KUKA KRL program: PickEsteira.src, PickEsteira.dat

--- PickEsteira.src ---
&ACCESS RVO1
&REL 243
&PARAM DISKPATH = KRC:\R1\Program\40293_Furukawa\Pick
DEF PickEsteira ( )
   ;FOLD INI;%{PE}
      ;FOLD BASISTECH INI
         GLOBAL INTERRUPT DECL 3 WHEN $STOPMESS==TRUE DO IR_STOPM ( )
         INTERRUPT ON 3
         BAS (#INITMOV,0 )
      ;ENDFOLD (BASISTECH INI)
      ;FOLD USER INI
         ;Make your modifications here

      ;ENDFOLD (USER INI)
   ;ENDFOLD (INI)
   ConfGarra_nowait()

   ;FOLD CONFIGURACOES DE MOVIMENTO
      $VEL.CP = 2.5
      $ACC.CP = 8
      $APO.CVEL = 80
      $APO.CPTP = 80
      $APO.CDIS = 20
      ;Base e Tool
      $TOOL = TOOL_DATA[1]
      $BASE = $NULLFRAME
   ;ENDFOLD

   ;configura o mesmo X  e Y do Xpick_esteira_1
   Xpick_esteira_2.X = Xpick_esteira_1.X
   Xpick_esteira_3.X = Xpick_esteira_1.X

   Xpick_esteira_2.Z = Xpick_esteira_1.Z
   Xpick_esteira_3.Z = Xpick_esteira_1.Z

   SWITCH PickOp
      CASE 1
         XAPP1PICK = Xpick_esteira_1
         XSAIPICK  = Xpick_esteira_1
      CASE 2
         XAPP1PICK = Xpick_esteira_2
         XSAIPICK  = Xpick_esteira_3
   ENDSWITCH

   XAPP1PICK.Z = ALTURAPICK
   XSAIPICK.Z  = ALTURAPICK

   ;APROXIMA TOPO
   PTP XAPP1PICK C_DIS

   ;CONFIGURA GARRA
   AbreGarra()
   ;ConfGarra_Wait()

   ;PONTO DE PICK
   SWITCH PickOp
      CASE 1
         ;FOLD LIN pick_esteira_1 Vel=2 m/s CPDAT1 Tool[1]:GarraUniversal Base[0] ;%{PE}
            ;FOLD Parameters ;%{h}
               ;Params IlfProvider=kukaroboter.basistech.inlineforms.movement.old; Kuka.IsGlobalPoint=False; Kuka.PointName=pick_esteira_1; Kuka.BlendingEnabled=False; Kuka.MoveDataName=CPDAT1; Kuka.VelocityPath=2; Kuka.CurrentCDSetIndex=0; Kuka.MovementParameterFieldEnabled=True; IlfCommand=LIN
            ;ENDFOLD
            $BWDSTART = FALSE
            LDAT_ACT = LCPDAT1_esteira
            FDAT_ACT = Fpick_esteira_1
            BAS(#CP_PARAMS, 2.0)
            SET_CD_PARAMS (0)
            LIN Xpick_esteira_1
         ;ENDFOLD
      CASE 2
;FOLD LIN pick_esteira_2 CONT Vel=2 m/s CPDAT2 Tool[1]:GarraUniversal Base[0] ;%{PE}
;FOLD Parameters ;%{h}
;Params IlfProvider=kukaroboter.basistech.inlineforms.movement.old; Kuka.IsGlobalPoint=False; Kuka.PointName=pick_esteira_2; Kuka.BlendingEnabled=True; Kuka.MoveDataName=CPDAT2; Kuka.VelocityPath=2; Kuka.CurrentCDSetIndex=0; Kuka.MovementParameterFieldEnabled=True; IlfCommand=LIN
;ENDFOLD
$BWDSTART = FALSE
LDAT_ACT = LCPDAT2
FDAT_ACT = Fpick_esteira_2
BAS(#CP_PARAMS, 2.0)
SET_CD_PARAMS (0)
LIN Xpick_esteira_2 C_Dis C_Dis
;ENDFOLD

         ;FOLD LIN pick_esteira_3 Vel=2 m/s CPDAT2 Tool[1]:GarraUniversal Base[0] ;%{PE}
            ;FOLD Parameters ;%{h}
               ;Params IlfProvider=kukaroboter.basistech.inlineforms.movement.old; Kuka.IsGlobalPoint=False; Kuka.PointName=pick_esteira_3; Kuka.BlendingEnabled=False; Kuka.MoveDataName=CPDAT2; Kuka.VelocityPath=2; Kuka.CurrentCDSetIndex=0; Kuka.MovementParameterFieldEnabled=True; IlfCommand=LIN
            ;ENDFOLD
            $BWDSTART = FALSE
            LDAT_ACT = LCPDAT2_esteira
            FDAT_ACT = Fpick_esteira_3
            BAS(#CP_PARAMS, 2.0)
            SET_CD_PARAMS (0)
            LIN Xpick_esteira_3
         ;ENDFOLD
   ENDSWITCH

   ;Fecha Garra
   FechaGarra()

   ;LIN XSAIPICK C_DIS C_DIS

END

--- PickEsteira.dat ---
&ACCESS RVO1
&REL 243
&PARAM DISKPATH = KRC:\R1\Program\40293_Furukawa\Pick
DEFDAT  PICKESTEIRA PUBLIC
DECL E6POS XAPP1PICK={X 1810.00,Y 331.540924,Z 205.000,A -89.9933853,B -1.07773711E-14,C -180.000,S 2,T 2,E1 0.0,E2 0.0,E3 0.0,E4 0.0,E5 0.0,E6 0.0}
DECL E6POS XAPP2PICK={X 1839.57971,Y 331.540924,Z -199.292,A -89.9933853,B -1.07773711E-14,C -180.000,S 2,T 2,E1 0.0,E2 0.0,E3 0.0,E4 0.0,E5 0.0,E6 0.0}
DECL E6POS XPICK={X 1839.57971,Y -502.858154,Z -210.581238,A -89.9924088,B -1.01663605E-13,C -180.000,S 2,T 2,E1 0.0,E2 0.0,E3 0.0,E4 0.0,E5 0.0,E6 0.0}
DECL E6POS XSAIPICK={X 1810.00,Y 331.540924,Z 205.000,A -89.9933853,B -1.07773711E-14,C -180.000,S 2,T 2,E1 0.0,E2 0.0,E3 0.0,E4 0.0,E5 0.0,E6 0.0}
;pontos exportados de FURUKAWA
DECL LDAT LCPDAT1_esteira={VEL 2.00000,ACC 100.000,APO_DIST 500.000,APO_FAC 50.0000,AXIS_VEL 100.000,AXIS_ACC 100.000,ORI_TYP #VAR,CIRC_TYP #BASE,JERK_FAC 50.0000,GEAR_JERK 100.000,EXAX_IGN 0}
DECL LDAT LCPDAT2_esteira={VEL 2.00000,ACC 100.000,APO_DIST 500.000,APO_FAC 50.0000,AXIS_VEL 100.000,AXIS_ACC 100.000,ORI_TYP #VAR,CIRC_TYP #BASE,JERK_FAC 50.0000,GEAR_JERK 100.000,EXAX_IGN 0}
DECL GLOBAL E6POS Xpick_esteira_1={X 1810.00,Y 331.540924,Z -199.292,A -89.9933853,B -1.07773711E-14,C -180.000,S 2,T 2,E1 0.0,E2 0.0,E3 0.0,E4 0.0,E5 0.0,E6 0.0}
DECL FDAT Fpick_esteira_1={TOOL_NO 1,BASE_NO 0,IPO_FRAME #BASE,POINT2[] " "}
DECL E6POS Xpick_esteira_2={X 1810.00,Y -502.858154,Z -199.292,A -89.9924088,B -1.01663605E-13,C -180.000,S 2,T 2,E1 0.0,E2 0.0,E3 0.0,E4 0.0,E5 0.0,E6 0.0}
DECL FDAT Fpick_esteira_2={TOOL_NO 1,BASE_NO 0,IPO_FRAME #BASE,POINT2[] " "}
DECL E6POS Xpick_esteira_3={X 1810.00,Y -615.344604,Z -199.292,A -89.9924088,B 1.60590833E-13,C 180.000,S 2,T 2,E1 0.0,E2 0.0,E3 0.0,E4 0.0,E5 0.0,E6 0.0}
DECL FDAT Fpick_esteira_3={TOOL_NO 1,BASE_NO 0,IPO_FRAME #BASE,POINT2[] " "}
DECL LDAT LCPDAT2={VEL 2.00000,ACC 100.000,APO_DIST 500.000,APO_FAC 50.0000,AXIS_VEL 100.000,AXIS_ACC 100.000,ORI_TYP #VAR,CIRC_TYP #BASE,JERK_FAC 50.0000,GEAR_JERK 100.000,EXAX_IGN 0}
DECL MODULEPARAM_T LAST_TP_PARAMS={PARAMS[] "Kuka.PointName=pick_esteira_2; Kuka.FrameData.base_no=0; Kuka.FrameData.tool_no=1; Kuka.FrameData.ipo_frame=#BASE; Kuka.FrameData.point2=; Kuka.isglobalpoint=False; Kuka.MoveDataName=CPDAT2; Kuka.MovementData.apo_fac=50; Kuka.MovementData.apo_dist=500; Kuka.MovementData.axis_acc=100; Kuka.MovementData.axis_vel=100; Kuka.MovementData.circ_typ=#BASE; Kuka.MovementData.jerk_fac=50; Kuka.MovementData.ori_typ=#VAR; Kuka.MovementData.vel=2; Kuka.MovementData.acc=100; Kuka.MovementData.exax_ign=0; Kuka.VelocityPath=2; Kuka.BlendingEnabled=True; Kuka.CurrentCDSetIndex=0"}
ENDDAT
